Fanuc KAREL source: kb00045.KL

-- PROVISIONAL review KL for V1013-1; original PC SHA256 8ce05c6093980b651d50f447d775dc1ba602b47a74d82a2e148a89d2a820837f
-- Incomplete behavior may be omitted. Consult companion uncertainty JSON. Do not deploy.
PROGRAM KB00045
%NOLOCKGROUP
BEGIN
  -- UNRESOLVED_PC offsets 5-14; opcodes 3F,75
  -- UNRESOLVED_PC offsets 19-26; opcodes 9D,23
  -- UNRESOLVED_PC offsets 31-49; opcodes 27,22,2A,22,31
  -- UNRESOLVED_PC offsets 54-58; opcodes 7F
END KB00045
